(* PLC project  *)

CONFIGURATION Application
  RESOURCE Application ON PLC
    TASK SoftMotionPlanningTask(PRIORITY := 15);
  END_RESOURCE
END_CONFIGURATION
